Fanuc TP program (LS listing): S101_DR_T13N50.LS

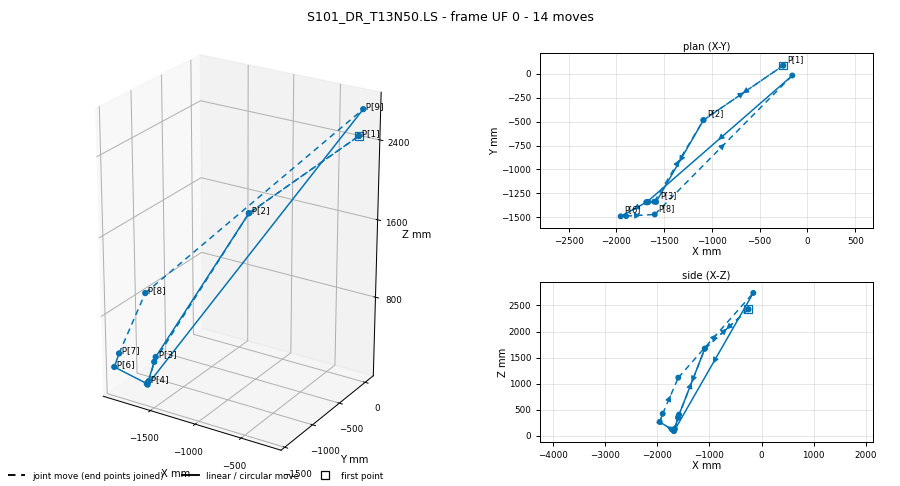
[picture p0: tool path of S101_DR_T13N50.LS in frame UF 0, 14 of 14 moves have a stored position in this frame; points joined in program order, loops and branches not executed]
/PROG  S101_DR_T13N50
/ATTR
OWNER		= MNEDITOR;
COMMENT		= "TL DRP TYP1 N50";
PROG_SIZE	= 3666;
CREATE		= DATE 21-06-09  TIME 06:40:36;
MODIFIED	= DATE 21-06-09  TIME 12:40:58;
FILE_NAME	= S101_DR_;
VERSION		= 0;
LINE_COUNT	= 121;
MEMORY_SIZE	= 4070;
PROTECT		= READ_WRITE;
STORAGE		= SHADOW;
TCD:  STACK_SIZE	= 0,
      TASK_PRIORITY	= 50,
      TIME_SLICE	= 0,
      BUSY_LAMP_OFF	= 0,
      ABORT_REQUEST	= 0,
      PAUSE_REQUEST	= 0;
DEFAULT_GROUP	= 1,*,*,*,*;
CONTROL_CODE	= 00000000 00000000;
/APPL
/MN
   1:  !******************************** ;
   2:  ! PATH - drop tool into N1=STA 70 ;
   3:  !******************************** ;
   4:  !* Robot ID: XXXXXR02B1 ;
   5:  !*    F-19XXXX ;
   6:  !* Line: XXXXXXXX ;
   7:  !* Platform: XX ;
   8:  !* Tool ID: TOOL xx ;
   9:  !* Program: S001_DR_TxxN3_R02 ;
  10:  !* Application: TOOL DROP ;
  11:  !******************************** ;
  12:  ! Author- Esys Automation ;
  13:  !******************************** ;
  14:   ;
  15:  !++++++++++++++++++++++++++++++++ ;
  16:  !ASSIGN PROGRAM PATH VALUES ;
  17:  !-------------------------------- ;
  18:  !Set Robot Tool and World UFrame ;
  19:  UTOOL_NUM=2 ;
  20:  UFRAME_NUM=0 ;
  21:  !++++++++++++++++++++++++++++++++ ;
  22:   ;
  23:  !******************************** ;
  24:  !BEGINNING OF PROGRAM PATH ;
  25:  !MOVE TO NEST 1 TOOL DROP ;
  26:  !******************************** ;
  27:   ;
  28:  !-------------------------------- ;
  29:  LBL[10:MOVE TO TL DRP] ;
  30:   ;
  31:  SET SEGMENT(50) ;
  32:  !SEG(50), Approach Tool Drop ;
  33:   ;
  34:J P[1] 100% CNT100    ;
  35:J P[2] 100% CNT100    ;
  36:   ;
  37:L P[3] 1000mm/sec CNT100    ;
  38:L P[4] 200mm/sec CNT25    ;
  39:   ;
  40:L P[5: Drop Tool] 50mm/sec FINE    ;
  41:   ;
  42:   ;
  43:  !-------------------------------- ;
  44:  LBL[20:UNLATCH TOOL] ;
  45:  UNLATCH TOOL    ;
  46:   ;
  47:  !ADD DISCONNECT COMMANDS ;
  48:  !ADD ALL EOAT DEVICES ;
  49:  !CALL EN_ARON(x) ;
  50:  !x = EOAT ENET Node # ;
  51:   ;
  52:  !If TL UNL Pass, Return Home ;
  53:  !If TL UNL Fail, Latch Tool, ;
  54:  !  MHFault, and Return Home ;
  55:  IF R[170]=1,JMP LBL[30] ;
  56:   ;
  57:  SELECT R[168]=7,JMP LBL[80] ;
  58:         ELSE,JMP LBL[99] ;
  59:   ;
  60:  !-------------------------------- ;
  61:  LBL[30:COMPLETE PATH] ;
  62:  !TL DRP COMPLETE. MOVE AWAY ;
  63:  !AND RETURN HOME ;
  64:   ;
  65:  !Set ATI Tool and World Frame ;
  66:  PAYLOAD[1] ;
  67:  UTOOL_NUM=14 ;
  68:  UFRAME_NUM=0 ;
  69:   ;
  70:  SET SEGMENT(51) ;
  71:  !SEG(51), Tool Drop Depart ;
  72:   ;
  73:L P[6] 50mm/sec FINE    ;
  74:   ;
  75:L P[7] 1000mm/sec CNT100    ;
  76:   ;
  77:J P[8] 100% CNT100    ;
  78:J P[9] 100% CNT100    ;
  79:   ;
  80:  ! Move To Home ;
  81:  JMP LBL[100] ;
  82:   ;
  83:  !-------------------------------- ;
  84:  LBL[80:UNLATCH FAULT] ;
  85:  !MOVE BACK TO HOME WITH TOOL ;
  86:  !on Reverse Path before Tool Drop ;
  87:   ;
  88:  !Set Payload= ATI ;
  89:  R[221]=1    ;
  90:  PAYLOAD[R[221]] ;
  91:   ;
  92:  UFRAME_NUM=0 ;
  93:  UTOOL_NUM=2 ;
  94:   ;
  95:  LATCH TOOL    ;
  96:   ;
  97:L P[14] 50mm/sec FINE    ;
  98:L P[10] 200mm/sec FINE    ;
  99:   ;
 100:J P[11] 100% CNT100    ;
 101:J P[12] 100% CNT100    ;
 102:J P[13] 100% CNT100    ;
 103:   ;
 104:  SET SEGMENT(63) ;
 105:  !SEG(63), Robot Move to Home ;
 106:   ;
 107:  R[132]=0    ;
 108:  GO[71]=0 ;
 109:   ;
 110:  ! Move To Home ;
 111:  JMP LBL[100] ;
 112:   ;
 113:  !-------------------------------- ;
 114:  LBL[99:ABORT PROGRAM] ;
 115:  MESSAGE[...] ;
 116:  MESSAGE[ABORT PROGRAM] ;
 117:  ABORT ;
 118:   ;
 119:  !-------------------------------- ;
 120:  LBL[100:END OF PROGRAM] ;
 121:  END ;
/POS
P[1]{
   GP1:
	UF : 0, UT : 2,		CONFIG : 'N U B, 0, 0, 0',
	X =  -253.309  mm,	Y =    88.383  mm,	Z =  2426.870  mm,
	W =   -93.331 deg,	P =     1.054 deg,	R =   122.429 deg
};
P[2]{
   GP1:
	UF : 0, UT : 2,		CONFIG : 'N U T, 0, 0, 0',
	X = -1089.020  mm,	Y =  -483.560  mm,	Z =  1671.145  mm,
	W =  -119.401 deg,	P =    -2.194 deg,	R =   112.860 deg
};
P[3]{
   GP1:
	UF : 0, UT : 2,		CONFIG : 'N U T, 0, 0, 0',
	X = -1584.026  mm,	Y = -1339.483  mm,	Z =   404.786  mm,
	W =  -161.490 deg,	P =      .518 deg,	R =    90.799 deg
};
P[4]{
   GP1:
	UF : 0, UT : 2,		CONFIG : 'N U T, 0, 0, 0',
	X = -1675.891  mm,	Y = -1343.409  mm,	Z =   112.875  mm,
	W =  -161.490 deg,	P =      .518 deg,	R =    90.799 deg
};
P[5:" Drop Tool"]{
   GP1:
	UF : 0, UT : 2,		CONFIG : 'N U T, 0, 0, 0',
	X = -1687.254  mm,	Y = -1343.718  mm,	Z =    96.307  mm,
	W =  -161.490 deg,	P =      .518 deg,	R =    90.799 deg
};
P[6:""]{
   GP1:
	UF : 0, UT : 14,		CONFIG : 'N U T, 0, 0, 0',
	X = -1955.045  mm,	Y = -1490.553  mm,	Z =   264.615  mm,
	W =  -159.945 deg,	P =      .151 deg,	R =    92.174 deg
};
P[7]{
   GP1:
	UF : 0, UT : 14,		CONFIG : 'N U T, 0, 0, 0',
	X = -1897.900  mm,	Y = -1487.967  mm,	Z =   421.300  mm,
	W =  -159.945 deg,	P =      .152 deg,	R =    92.174 deg
};
P[8]{
   GP1:
	UF : 0, UT : 14,		CONFIG : 'N U T, 0, 0, 0',
	X = -1598.294  mm,	Y = -1470.396  mm,	Z =  1114.792  mm,
	W =  -159.094 deg,	P =      .421 deg,	R =    91.998 deg
};
P[9]{
   GP1:
	UF : 0, UT : 14,		CONFIG : 'N U B, 0, 0, 0',
	X =  -158.400  mm,	Y =   -15.894  mm,	Z =  2741.103  mm,
	W =   -91.792 deg,	P =     -.357 deg,	R =   122.600 deg
};
P[10]{
   GP1:
	UF : 0, UT : 2,		CONFIG : 'N U T, 0, 0, 0',
	X = -1666.068  mm,	Y = -1340.792  mm,	Z =   128.711  mm,
	W =  -161.733 deg,	P =      .481 deg,	R =    90.252 deg
};
P[11]{
   GP1:
	UF : 0, UT : 2,		CONFIG : 'N U T, 0, 0, 0',
	X = -1603.494  mm,	Y = -1336.916  mm,	Z =   346.817  mm,
	W =  -161.727 deg,	P =      .345 deg,	R =    90.001 deg
};
P[12]{
   GP1:
	UF : 0, UT : 2,		CONFIG : 'N U T, 0, 0, 0',
	X = -1089.020  mm,	Y =  -483.560  mm,	Z =  1671.145  mm,
	W =  -119.401 deg,	P =    -2.194 deg,	R =   112.860 deg
};
P[13]{
   GP1:
	UF : 0, UT : 2,		CONFIG : 'N U B, 0, 0, 0',
	X =  -253.309  mm,	Y =    88.384  mm,	Z =  2426.870  mm,
	W =   -93.331 deg,	P =     1.054 deg,	R =   122.429 deg
};
P[14]{
   GP1:
	UF : 0, UT : 2,		CONFIG : 'N U T, 0, 0, 0',
	X = -1681.218  mm,	Y = -1341.312  mm,	Z =    86.634  mm,
	W =  -161.733 deg,	P =      .481 deg,	R =    90.252 deg
};
/END
